Staubli VAL3: cvIn.dtx

bool bClockEnabled = true
bool bEnableQueuing = true
bool bInit = true
public bool bLOG = true
public bool bLinear = true
bool bLockQueueAcces
bool bResetConv
public bool bUseUserCenter
public bool bUseUserLimit
dio doClock = {link=BasicIO-1\%Q0}
public frame fConveyor = {x=365.904087, y=326.91934, z=-82.602337, rx=-0.010861, ry=-0.059106, rz=0.004608, fatherId=world[0]}
public frame fDetection = {x=392.598601, y=461.346273, z=-82.976862, rx=0.205045, ry=0.617271, rz=0.011036, fatherId=world[0]}
num nA1 = -1.427414
num nA2 = -1.428787
num nAddedToQueue
num nB1
num nB2 = 436.58822
num nBoundaryDwn
num nBoundaryUp
public num nBufferSize = 100
public num nCalibratedDist
num nCalibratedID = -99
public num nClockPeriod = 210
public num nConveyorSpeed
num nDEFAULTID = -99
num nDETECT_OVR = 11
public num nDetection2Rob = 945.961992
public num nENCRESOLUTION = 2000
public num nENCSCALEFACTOR = 0.7207
num nEncLatchedVal[100]
  [0] = 10423725.84
  [1] = 10423725.84
  [2] = 10424018.43
  [3] = 10424018.43
  [4] = 10425772.17
  [5] = 10426066.875
  [6] = 10426359.285
  [7] = 10426359.285
  [8] = 10434839.175
  [9] = 10434839.175
  [10] = 10436885.46
  [11] = 10437177.96
  [12] = 10437177.96
  [13] = 10437470.595
  [14] = 10394182.305
  [15] = 10394474.85
  [16] = 10394474.85
  [17] = 10394767.35
  [18] = 10394767.35
  [19] = 10395059.58
  [20] = 10395059.58
  [21] = 10395351.945
  [22] = 10395351.945
  [23] = 10395644.355
  [24] = 10395644.355
  [25] = 10395935.19
  [26] = 10395935.19
  [27] = 10396230.165
  [28] = 10396230.165
  [29] = 10396522.8
  [30] = 10396522.8
  [31] = 10396817.37
  [32] = 10396817.37
  [33] = 10396817.37
  [34] = 10397109.96
  [35] = 10397109.96
  [36] = 10397109.96
  [37] = 10397402.55
  [38] = 10397402.55
  [39] = 10397402.55
  [40] = 10397694.87
  [41] = 10397694.87
  [42] = 10397694.87
  [43] = 10397987.1
  [44] = 10397987.1
  [45] = 10397987.1
  [46] = 10398281.625
  [47] = 10398281.625
  [48] = 10398281.625
  [49] = 10398574.35
  [50] = 10398574.35
  [51] = 10398574.35
  [52] = 10398865.095
  [53] = 10398865.095
  [54] = 10398865.095
  [55] = 10399157.82
  [56] = 10399157.82
  [57] = 10399157.82
  [58] = 10399452.57
  [59] = 10399452.57
  [60] = 10399452.57
  [61] = 10399745.25
  [62] = 10399745.25
  [63] = 10399745.25
  [64] = 10400037.84
  [65] = 10400037.84
  [66] = 10400037.84
  [67] = 10400330.295
  [68] = 10400330.295
  [69] = 10400330.295
  [70] = 10400622.795
  [71] = 10400917.32
  [72] = 10401209.82
  [73] = 10408224.06
  [74] = 10408516.335
  [75] = 10408516.335
  [76] = 10408808.745
  [77] = 10410563.925
  [78] = 10410856.83
  [79] = 10411149.555
  [80] = 10412614.215
  [81] = 10412906.715
  [82] = 10412906.715
  [83] = 10413199.35
  [84] = 10414953.135
  [85] = 10414953.135
  [86] = 10415245.32
  [87] = 10415537.82
  [88] = 10416996.54
  [89] = 10417289.175
  [90] = 10417289.175
  [91] = 10417581.855
  [92] = 10419335.1
  [93] = 10419627.825
  [94] = 10419627.825
  [95] = 10419627.825
  [96] = 10421675.46
  [97] = 10421675.46
  [98] = 10421675.46
  [99] = 10421968.005
num nErrVal[4]
public num nFirDelay = 0.004
public num nFirOrdre = 20
num nFirTime = 0.04
num nIdxCalib
num nIdxPull = 14
num nIdxPush = 14
public num nLatchLockDist
num nNumbOfUser[100]
num nPUSH_NEGATIVE = 10
public num nPosMatchTol = 50
num nQueueID[100]
  [0] = -1
  [1] = -1
  [2] = -1
  [3] = -1
  [4] = -1
  [5] = -1
  [6] = -1
  [7] = -1
  [8] = -1
  [9] = -1
  [10] = -1
  [11] = -1
  [12] = -1
  [13] = -1
  [14] = -1
  [15] = -1
  [16] = -1
  [17] = -1
  [18] = -1
  [19] = -1
  [20] = -1
  [21] = -1
  [22] = -1
  [23] = -1
  [24] = -1
  [25] = -1
  [26] = -1
  [27] = -1
  [28] = -1
  [29] = -1
  [30] = -1
  [31] = -1
  [32] = -1
  [33] = -1
  [34] = -1
  [35] = -1
  [36] = -1
  [37] = -1
  [38] = -1
  [39] = -1
  [40] = -1
  [41] = -1
  [42] = -1
  [43] = -1
  [44] = -1
  [45] = -1
  [46] = -1
  [47] = -1
  [48] = -1
  [49] = -1
  [50] = -1
  [51] = -1
  [52] = -1
  [53] = -1
  [54] = -1
  [55] = -1
  [56] = -1
  [57] = -1
  [58] = -1
  [59] = -1
  [60] = -1
  [61] = -1
  [62] = -1
  [63] = -1
  [64] = -1
  [65] = -1
  [66] = -1
  [67] = -1
  [68] = -1
  [69] = -1
  [70] = -1
  [71] = -1
  [72] = -1
  [73] = -1
  [74] = -1
  [75] = -1
  [76] = -1
  [77] = -1
  [78] = -1
  [79] = -1
  [80] = -1
  [81] = -1
  [82] = -1
  [83] = -1
  [84] = -1
  [85] = -1
  [86] = -1
  [87] = -1
  [88] = -1
  [89] = -1
  [90] = -1
  [91] = -1
  [92] = -1
  [93] = -1
  [94] = -1
  [95] = -1
  [96] = -1
  [97] = -1
  [98] = -1
  [99] = -1
num nStatus
num nSysCycleTime = 0.002
num nTmpEncLatched[10]
  [0] = 10437470.595
  [1] = 10437470.595
  [2] = 10437177.96
  [3] = 10424018.43
num nTmpID[10]
  [0] = 1
  [1] = 1
  [2] = 1
  [3] = 1
public num nTrackWinHeight = 500
num nWinDownStream
num nWinUpStream
pointRs pObjectRS = {fatherId=world[0]}
pointRx pObject = {fatherId=world[0]}
public string sClockSigName = "bOut0"
string sConvNum = "CNV0"
public string sConveyorName = "cvIn"
public string sDetectionLib = "PointGrey"
public string sDwnLimSigName = "none"
public string sEncoderLib = "D_ABZ_00"
string sErrMsgList[12]
  [0] = "Success"
  [1] = "No object available (ID=*)"
  [3] = "The encoder library is not started yet."
  [4] = "The detection library is not started yet."
  [6] = "Run-time error from Conveyor library in task called *\../*. Error code is *"
  [7] = "Run-time error from Encoder library. Error code is *"
  [8] = "Run-time error from Detection library. Error code is *"
  [10] = "Warning, object with negative ID cannot be pushed into conveyor's queue"
  [11] = "Warning, detection overrun."
string sErrorMessage = "No message pending"
public string sGeometryLib = "GeometryRS"
string sMsg
string sTASK[3]
  [0] = "conveyor"
  [1] = "encoder"
  [2] = "detect"
public string sUpLimSigName = "none"
trsf trBoundaryDwn[2]
  [0] = {x=305.565702, rx=-179.989134, ry=-0.059105, rz=88.399965}
  [1] = {x=118.089887, y=267.862957, z=0.515773, rx=-179.989134, ry=-0.059105, rz=65.426002}
trsf trBoundaryUp[2]
  [0] = {rx=-179.989134, ry=-0.059105, rz=58.053225}
  [1] = {x=-187.656083, y=267.862957, rx=-179.989134, ry=-0.059105, rz=32.698528}
trsf trDEFAULT = {x=5, y=4, z=3, rx=2, ry=1}
trsf trDetectedCoord[100]
  [0] = {x=-58, y=-27, rz=74.4}
  [1] = {x=-153, y=-23, rz=68.3}
  [2] = {x=-84, y=-11, rz=89.5}
  [3] = {x=-176, y=-4, rz=87.7}
  [4] = {x=-182, y=-17, rz=84.6}
  [5] = {x=-86, y=-18, rz=92}
  [6] = {x=9, y=-21, rz=82.8}
  [7] = {x=-90, y=-8, rz=101.2}
  [8] = {x=7, y=-17, rz=85.8}
  [9] = {x=-102, y=-29, rz=84.2}
  [10] = {x=-82, y=-12, rz=80.8}
  [11] = {x=9, y=-15, rz=79.8}
  [12] = {x=-90, y=-15, rz=86.9}
  [13] = {x=-13, y=-18, rz=76.8}
  [14] = {x=-156, y=-10, rz=60}
  [15] = {x=-8, y=-21, rz=60.4}
  [16] = {x=-156, y=-9, rz=58.6}
  [17] = {x=-8, y=-16, rz=64.2}
  [18] = {x=-156, y=-13, rz=62.7}
  [19] = {x=-10, y=-13, rz=63.8}
  [20] = {x=-156, y=-13, rz=62.9}
  [21] = {x=-9, y=-16, rz=63.2}
  [22] = {x=-155, y=-13, rz=62.4}
  [23] = {x=-8, y=-22, rz=63}
  [24] = {x=-156, y=-12, rz=62}
  [25] = {x=-4, y=-4, rz=64.5}
  [26] = {x=-156, y=-11, rz=61.5}
  [27] = {x=-9, y=-13, rz=63.1}
  [28] = {x=-156, y=-12, rz=62.1}
  [29] = {x=-9, y=-12, rz=63.4}
  [30] = {x=-155, y=-13, rz=62.6}
  [31] = {x=125, y=-7, rz=73}
  [32] = {x=-7, y=-23, rz=61.7}
  [33] = {x=-155, y=-11, rz=60.4}
  [34] = {x=112, y=33, rz=71.2}
  [35] = {x=-10, y=-8, rz=63.5}
  [36] = {x=-155, y=-12, rz=62.1}
  [37] = {x=121, y=27, rz=71.8}
  [38] = {x=-8, y=-13, rz=63.1}
  [39] = {x=-156, y=-12, rz=61.2}
  [40] = {x=109, y=47, rz=70.6}
  [41] = {x=-10, y=-1, rz=63.3}
  [42] = {x=-155, y=-10, rz=60.8}
  [43] = {x=108, y=46, rz=70.7}
  [44] = {x=-9, y=-4, rz=64.2}
  [45] = {x=-155, y=-11, rz=61.2}
  [46] = {x=113, y=58, rz=72.2}
  [47] = {x=-10, y=2, rz=63.1}
  [48] = {x=-154, y=-8, rz=59.2}
  [49] = {x=116, y=58, rz=72.9}
  [50] = {x=-10, y=3, rz=62.1}
  [51] = {x=-153, y=-7, rz=59}
  [52] = {x=113, y=58, rz=71.3}
  [53] = {x=-12, y=1, rz=61.7}
  [54] = {x=-153, y=-9, rz=59.7}
  [55] = {x=112, y=58, rz=72.8}
  [56] = {x=-10, y=1, rz=63.2}
  [57] = {x=-153, y=-10, rz=60.4}
  [58] = {x=111, y=42, rz=70.7}
  [59] = {x=-9, y=-6, rz=62.7}
  [60] = {x=-155, y=-11, rz=60.5}
  [61] = {x=120, y=20, rz=71.7}
  [62] = {x=-9, y=-14, rz=62}
  [63] = {x=-155, y=-11, rz=60.5}
  [64] = {x=133, y=13, rz=83.5}
  [65] = {x=-6, y=-7, rz=61.4}
  [66] = {x=-155, y=-12, rz=61}
  [67] = {x=103, y=20, rz=77.5}
  [68] = {x=-18, y=-8, rz=65.2}
  [69] = {x=-169, y=-1, rz=61.9}
  [70] = {x=-147, y=-75, rz=105.8}
  [71] = {x=-142, y=-84, rz=107.8}
  [72] = {x=-132, y=-84, rz=98.3}
  [73] = {x=-174, y=-15, rz=97.3}
  [74] = {x=-65, y=-21, rz=102.4}
  [75] = {x=-168, y=-8, rz=92.1}
  [76] = {x=-67, y=-1, rz=82}
  [77] = {x=-83, y=-24, rz=70}
  [78] = {x=-18, y=-42, rz=76.5}
  [79] = {x=1, y=-13, rz=80.3}
  [80] = {x=-226, y=-61, rz=67}
  [81] = {x=-88, y=-23, rz=96.8}
  [82] = {x=-192, y=-7, rz=84.6}
  [83] = {x=-102, y=-16, rz=79.7}
  [84] = {x=-58, y=-16, rz=104.2}
  [85] = {x=-146, y=-55, rz=103.9}
  [86] = {x=-66, y=-19, rz=72.8}
  [87] = {x=24, y=-15, rz=78}
  [88] = {x=-173, y=-2, rz=86.1}
  [89] = {x=-53, y=-35, rz=94.3}
  [90] = {x=-181, y=3, rz=87.7}
  [91] = {x=-84, y=-3, rz=91.1}
  [92] = {x=-62, y=-8, rz=83.9}
  [93] = {x=40, y=-35, rz=102.5}
  [94] = {x=-65, y=-49, rz=93}
  [95] = {x=-169, y=-7, rz=95}
  [96] = {x=33, y=-20, rz=89.3}
  [97] = {x=-59, y=-21, rz=90.9}
  [98] = {x=-158, y=-9, rz=85.4}
  [99] = {x=-69, y=-3, rz=80}
trsf trTmp[10]
  [0] = {x=118, y=-13, rz=82}
  [1] = {x=-13, y=-18, rz=76.8}
  [2] = {x=-90, y=-15, rz=86.9}
  [3] = {x=-176, y=-4, rz=87.7}
